// TIA Portal V16 export
// export: Created 2020-09-25T08:26:19.1199448Z, ExportSetting WithDefaults, DisplayName Totally Integrated Automation Portal, DisplayVersion V16 Update 2, DisplayName TIA Portal Version Control Interface, DisplayVersion V16 Update 2, DisplayName TIA Portal Openness, DisplayVersion V16 Update 2, DisplayName STEP 7 Professional, DisplayVersion V16 Update 2, DisplayName STEP 7 Safety, DisplayVersion V16, DisplayName WinCC Advanced, DisplayVersion V16 Update 2
DATA_BLOCK "Baustein_2_DB"   // DB2
VERSION : 0.1
// stored: AutoNumber true, InstanceOfName Baustein_2, InstanceOfType FB
"Baustein_2"
   // VAR_INPUT
   //    input1 : Bool;
   //    input2 : Bool;
   // END_VAR
BEGIN
END_DATA_BLOCK
